ABB RobotStudio station: Exercise1.rspag

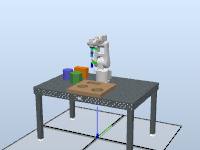
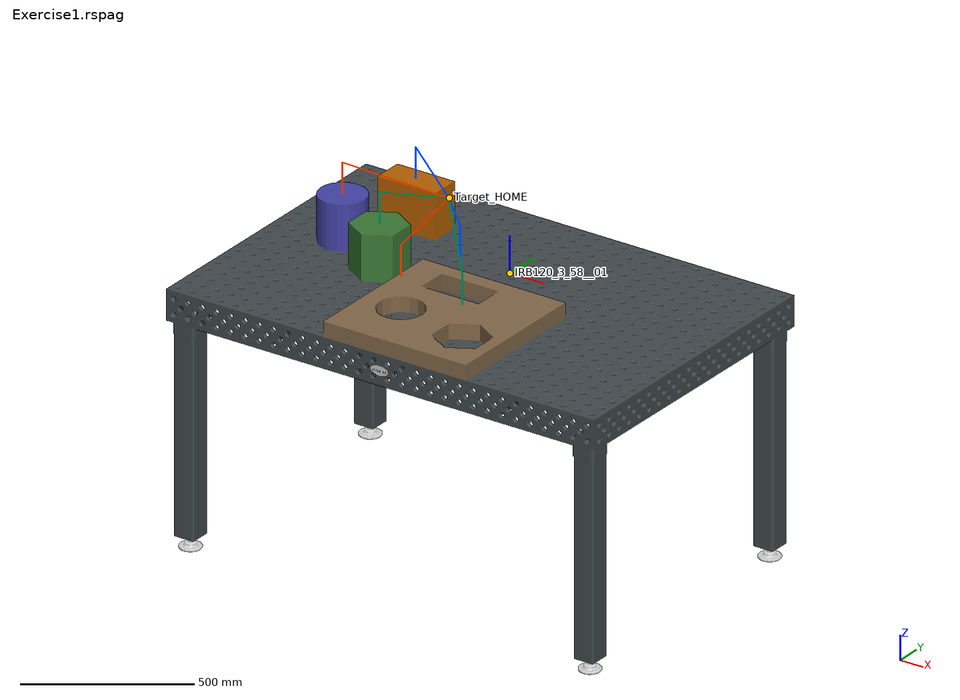
[picture v1: parts stored in the station drawn from their meshes, with robot base, taught points and paths (robot models come from the ABB library and are not in the file)]
--- station ---
Station Ex1_complete (saved by RobotStudio 21.4.9700.0)
Controller Controller1, task T_ROB1: task frame (RAPID world) sits at (0, 150, 830) mm, rotated rx 0 ry 0 rz -90 deg in the station
Controller Controller1
  mechanical unit ROB_1: IRB120_3_58__01, 6 joints, base frame (0, 0, 0) mm
Layout (positions relative to the parent item):
  - table [part] at (-200, -500, 830) mm, size 500 x 500 x 50 mm
  - object_1 [part] at (-600, -150, 830) mm, size 200 x 100 x 150 mm
  - object_2 [part] at (-650, -150, 830) mm, size 149.5 x 149.7 x 150 mm
  - siegmund_1500_1000 [part], size 1500 x 1010.3 x 830 mm
  - object_11 [part] at (-200, -500, 830) mm, size 200 x 100 x 150 mm
  - object_22 [part] at (-200, -500, 830) mm, size 149.5 x 149.7 x 150 mm
  - object_33 [part] at (-200, -500, 830) mm, size 155.5 x 179.5 x 150 mm
  - smc_gripper [mechanism, from Cvičení\smc_gripper.rslib] at (0, -152.6, 1388) mm, rotated rx 180 ry 0.47 rz 90 deg
  - IRB120_3_58__01 [mechanism, from Robots\IRB120_3_58_G_01.rslib] at (0, 150, 830) mm, rotated rx 0 ry 0 rz -90 deg; joint values [0, 0, 0, 0, 1.5625, 0] (rad or m)
  - object_3 [part] at (-700, -200, 830) mm, size 155.5 x 179.5 x 150 mm
  - Positioner_OBJ3 [smart component, from Components\Positioner.rslib]
      properties: Object=object_3; Position=[-0.7 -0.2 0.83]; Orientation=[0 0 0]; Reference=Global; ReferenceObject=(none)
  - Attacher_OBJ3 [smart component, from Components\Attacher.rslib]
      properties: Parent=smc_gripper; Flange=0; Child=object_3; Mount=false; Offset=[0 0 0]; Orientation=[0 0 0]
  - Detacher_OBJ3 [smart component, from Components\Detacher.rslib]
      properties: Child=object_3; KeepPosition=true
  - Positioner_OBJ2 [smart component, from Components\Positioner.rslib]
      properties: Object=object_2; Position=[-0.65 -0.15 0.83]; Orientation=[0 0 0]; Reference=Global; ReferenceObject=(none)
  - Positioner_OBJ1 [smart component, from Components\Positioner.rslib]
      properties: Object=object_1; Position=[-0.6 -0.15 0.83]; Orientation=[0 0 0]; Reference=Global; ReferenceObject=(none)
  - Attacher_OBJ1 [smart component, from Components\Attacher.rslib]
      properties: Parent=smc_gripper; Flange=0; Child=object_1; Mount=false; Offset=[0 0 0]; Orientation=[0 0 0]
  - Detacher_OBJ1 [smart component, from Components\Detacher.rslib]
      properties: Child=object_1; KeepPosition=true
  - Attacher_OBJ2 [smart component, from Components\Attacher.rslib]
      properties: Parent=smc_gripper; Flange=0; Child=object_2; Mount=false; Offset=[0 0 0]; Orientation=[0 0 0]
  - Detacher_OBJ2 [smart component, from Components\Detacher.rslib]
      properties: Child=object_2; KeepPosition=true
Attachment: smc_gripper is attached to IRB120_3_58__01 / Link6
Station signals: DI DI_POS_OBJ
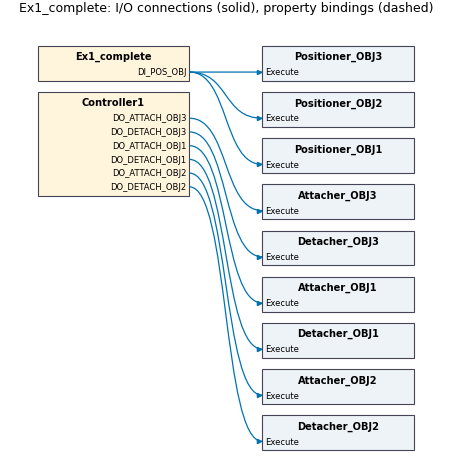
Station logic (signal -> signal, property => property):
  Ex1_complete.DI_POS_OBJ -> Positioner_OBJ3.Execute
  Ex1_complete.DI_POS_OBJ -> Positioner_OBJ2.Execute
  Ex1_complete.DI_POS_OBJ -> Positioner_OBJ1.Execute
  Controller1.DO_ATTACH_OBJ3 -> Attacher_OBJ3.Execute
  Controller1.DO_DETACH_OBJ3 -> Detacher_OBJ3.Execute
  Controller1.DO_ATTACH_OBJ1 -> Attacher_OBJ1.Execute
  Controller1.DO_DETACH_OBJ1 -> Detacher_OBJ1.Execute
  Controller1.DO_ATTACH_OBJ2 -> Attacher_OBJ2.Execute
  Controller1.DO_DETACH_OBJ2 -> Detacher_OBJ2.Execute

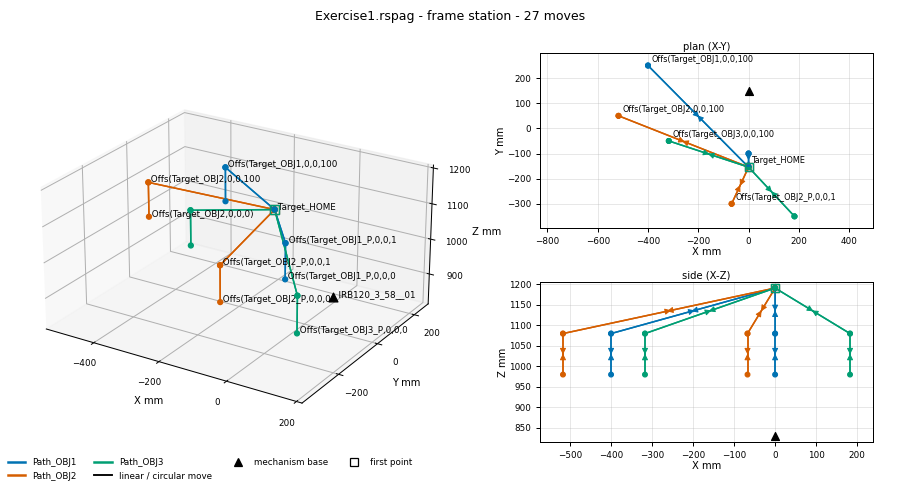
[picture p0: tool path of Exercise1.rspag in frame station, 27 of 27 moves have a stored position in this frame; points joined in program order, loops and branches not executed]
--- Backups/Controller1/RAPID/TASK1/PROGMOD/CalibData.mod ---
MODULE CalibData
    PERS tooldata smc_gripper:=[TRUE,[[0,0.004,197.001],[1,0,0,0]],[1,[0.207,-0.496,71.18],[1,0,0,0],0,0,0]];
ENDMODULE

--- Backups/Controller1/RAPID/TASK1/PROGMOD/Module1.mod ---
MODULE Module1
    CONST robtarget Target_HOME:=[[304.223785172,0.004,361.008191983],[0.004133449,0,0.999991457,0],[0,0,0,0],[9E+09,9E+09,9E+09,9E+09,9E+09,9E+09]];
    CONST robtarget Target_OBJ1:=[[-100,-400,150],[0,0.707106781,0.707106781,0],[-2,0,-1,0],[9E+09,9E+09,9E+09,9E+09,9E+09,9E+09]];
    CONST robtarget Target_OBJ1_P:=[[250,0,150],[0,0.707106781,0.707106781,0],[0,0,0,0],[9E+09,9E+09,9E+09,9E+09,9E+09,9E+09]];
    CONST robtarget Target_OBJ2:=[[100,-517.298,150],[0,0.707106781,0.707106781,0],[0,0,0,0],[9E+09,9E+09,9E+09,9E+09,9E+09,9E+09]];
    CONST robtarget Target_OBJ2_P:=[[450,-67.298,150],[0,0.707106781,0.707106781,0],[0,0,0,0],[9E+09,9E+09,9E+09,9E+09,9E+09,9E+09]];
    CONST robtarget Target_OBJ3:=[[200,-317.298,150],[0,0.707106781,0.707106781,0],[0,0,0,0],[9E+09,9E+09,9E+09,9E+09,9E+09,9E+09]];
    CONST robtarget Target_OBJ3_P:=[[500,182.702,150],[0,0.707106781,0.707106781,0],[0,0,1,0],[9E+09,9E+09,9E+09,9E+09,9E+09,9E+09]];
!***********************************************************
    ! Description: Exercise 1 - complete
    !
    ! Author: Karolina Kovarova
    !
!***********************************************************
    PROC main()
        Path_OBJ3;
        Path_OBJ2;
        Path_OBJ1;
    ENDPROC

    PROC Path_OBJ1()
        MoveL Target_HOME,v200,fine,smc_gripper\WObj:=wobj0;

        MoveL Offs(Target_OBJ1, 0, 0, 100),v200,fine,smc_gripper\WObj:=wobj0;
        MoveL Offs(Target_OBJ1, 0, 0, 0),v200,fine,smc_gripper\WObj:=wobj0;
        waitTime 0.1;
        PulseDO DO_ATTACH_OBJ1;
        waitTime 0.1;
        MoveL Offs(Target_OBJ1, 0, 0, 100),v200,fine,smc_gripper\WObj:=wobj0;

        MoveL Target_HOME,v200,fine,smc_gripper\WObj:=wobj0;

        MoveL Offs(Target_OBJ1_P, 0, 0, 100),v200,fine,smc_gripper\WObj:=wobj0;
        MoveL Offs(Target_OBJ1_P, 0, 0, 0),v200,fine,smc_gripper\WObj:=wobj0;
        waitTime 0.1;
        PulseDO DO_DETACH_OBJ1;
        waitTime 0.1;
        MoveL Offs(Target_OBJ1_P, 0, 0, 100),v200,fine,smc_gripper\WObj:=wobj0;

        MoveL Target_HOME,v200,fine,smc_gripper\WObj:=wobj0;
    ENDPROC

    PROC Path_OBJ2()
        MoveL Target_HOME,v200,fine,smc_gripper\WObj:=wobj0;

        MoveL Offs(Target_OBJ2, 0, 0, 100),v200,fine,smc_gripper\WObj:=wobj0;
        MoveL Offs(Target_OBJ2, 0, 0, 0),v200,fine,smc_gripper\WObj:=wobj0;
        waitTime 0.1;
        PulseDO DO_ATTACH_OBJ2;
        waitTime 0.1;
        MoveL Offs(Target_OBJ2, 0, 0, 100),v200,fine,smc_gripper\WObj:=wobj0;

        MoveL Target_HOME,v200,fine,smc_gripper\WObj:=wobj0;

        MoveL Offs(Target_OBJ2_P, 0, 0, 100),v200,fine,smc_gripper\WObj:=wobj0;
        MoveL Offs(Target_OBJ2_P, 0, 0, 0),v200,fine,smc_gripper\WObj:=wobj0;
        waitTime 0.1;
        PulseDO DO_DETACH_OBJ2;
        waitTime 0.1;
        MoveL Offs(Target_OBJ2_P, 0, 0, 100),v200,fine,smc_gripper\WObj:=wobj0;

        MoveL Target_HOME,v200,fine,smc_gripper\WObj:=wobj0;
    ENDPROC

    PROC Path_OBJ3()
        MoveL Target_HOME,v200,fine,smc_gripper\WObj:=wobj0;

        MoveL Offs(Target_OBJ3, 0, 0, 100),v200,fine,smc_gripper\WObj:=wobj0;
        MoveL Offs(Target_OBJ3, 0, 0, 0),v200,fine,smc_gripper\WObj:=wobj0;
        waitTime 0.1;
        PulseDO DO_ATTACH_OBJ3;
        waitTime 0.1;
        MoveL Offs(Target_OBJ3, 0, 0, 100),v200,fine,smc_gripper\WObj:=wobj0;

        MoveL Target_HOME,v200,fine,smc_gripper\WObj:=wobj0;

        MoveL Offs(Target_OBJ3_P, 0, 0, 100),v200,fine,smc_gripper\WObj:=wobj0;
        MoveL Offs(Target_OBJ3_P, 0, 0, 0),v200,fine,smc_gripper\WObj:=wobj0;
        waitTime 0.1;
        PulseDO DO_DETACH_OBJ3;
        waitTime 0.1;
        MoveL Offs(Target_OBJ3_P, 0, 0, 100),v200,fine,smc_gripper\WObj:=wobj0;

        MoveL Target_HOME,v200,fine,smc_gripper\WObj:=wobj0;
    ENDPROC
ENDMODULE

--- Backups/Controller1/SYSPAR/EIO.cfg ---
EIO:CFG_1.0:6:1::
#
EIO_SIGNAL:

      -Name "DO_ATTACH_OBJ1" -SignalType "DO"

      -Name "DO_DETACH_OBJ1" -SignalType "DO"

      -Name "DO_ATTACH_OBJ2" -SignalType "DO"

      -Name "DO_DETACH_OBJ2" -SignalType "DO"

      -Name "DO_ATTACH_OBJ3" -SignalType "DO"

      -Name "DO_DETACH_OBJ3" -SignalType "DO"
